// Mitsubishi GX Works2 project: CODIGO BÁSICO   PLC: FX3U/FX3UC
// Configuração Modbus RTU

PROGRAM MAIN
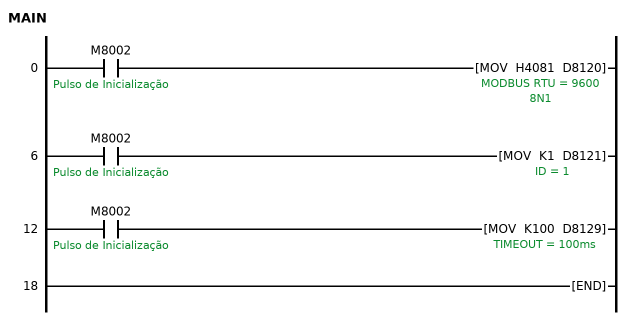
0     LD      M8002  ; Pulso de Inicialização
      MOV     H4081 D8120  ; MODBUS RTU = 9600 8N1
6     LD      M8002  ; Pulso de Inicialização
      MOV     K1 D8121  ; ID = 1
12    LD      M8002  ; Pulso de Inicialização
      MOV     K100 D8129  ; TIMEOUT = 100ms
18    END
END_PROGRAM

// device comments not shown above
X000  ; DIGITAL ENTRADA 0
X001  ; ENTRADA DIGITAL 1
Y000  ; RELE 0
Y001  ; RELE 1
Y002  ; RELE 2
M0  ; VARIAVEL DE MEMORIA 0
M1  ; VARIAVEL DE MEMORIA 1
M2  ; VARIAVEL DE MEMORIA 2
D0  ; REGISTRO 0
D1  ; LEITURA 1
D2  ; ENCHE O TANQUE
D3  ; ESVAZIA O TANQUE
